FUNCTION_BLOCK FB_HNHTMachineSystem
VAR_INPUT
END_VAR
VAR_OUTPUT
END_VAR
VAR
END_VAR

END_FUNCTION_BLOCK

(* stored: Version 1.1.0.1, ProductVersion 3.1.4024.10
   POU FB_HNHTMachineSystem: Id {a07e4849-9881-441f-b859-bc1231e9abc7}, SpecialFunc None *)
